FUNCTION_BLOCK LinearDA (* Basic Function Block Type *)
  (* Standard: 61499-2 *)
  (* Version 0.0, 12/23/2020, midhu, nxtControl GmbH, Template *)
  PACKAGE Main;
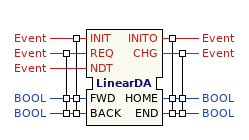
  EVENT_INPUT
    INIT WITH FWD, BACK;
    REQ WITH FWD, BACK; (* Initialization Request *)
    NDT; (* Non deterministic transition *)
  END_EVENT
  EVENT_OUTPUT
    INITO WITH HOME, END;
    CHG WITH HOME, END; (* Initialization Confirm *)
  END_EVENT
  VAR_INPUT
    FWD : BOOL; (* Input event qualifier *)
    BACK : BOOL;
  END_VAR
  VAR_OUTPUT
    HOME : BOOL; (* Output event qualifier *)
    END : BOOL;
  END_VAR
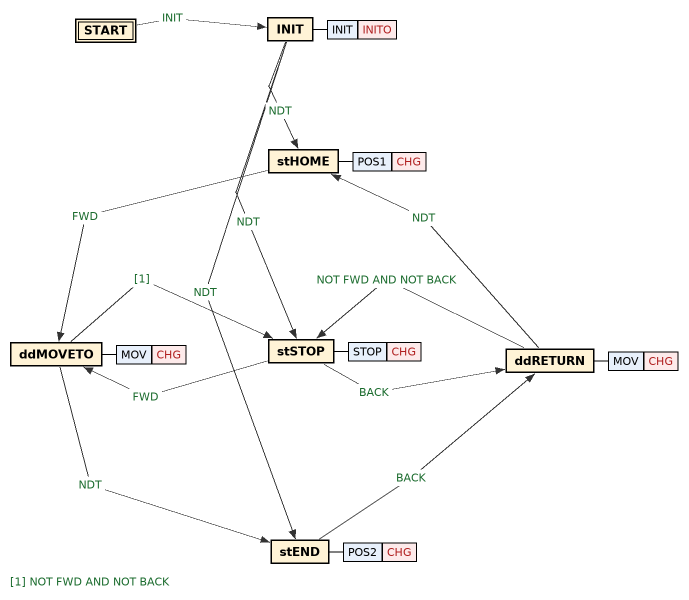
  EC_STATES
    START; (* Initial State *)
    INIT : INIT -> INITO; (* Initialization *)
    stHOME : POS1 -> CHG;
    stEND : POS2 -> CHG;
    ddMOVETO : MOV -> CHG;
    ddRETURN : MOV -> CHG;
    stSTOP : STOP -> CHG;
  END_STATES
  EC_TRANSITIONS
    START TO INIT := INIT;
    INIT TO stHOME := NDT;
    stHOME TO ddMOVETO := FWD;
    stEND TO ddRETURN := BACK;
    ddMOVETO TO stEND := NDT;
    ddRETURN TO stHOME := NDT;
    ddRETURN TO stSTOP := NOT FWD AND NOT BACK;
    stSTOP TO ddRETURN := BACK;
    stSTOP TO ddMOVETO := FWD;
    ddMOVETO TO stSTOP := NOT FWD AND NOT BACK;
    INIT TO stSTOP := NDT;
    INIT TO stEND := NDT;
  END_TRANSITIONS
  ALGORITHM INIT IN ST: (* Initialization algorithm *)
HOME  :=TRUE;
END   :=FALSE;
  END_ALGORITHM
  ALGORITHM POS1 IN ST:
HOME  :=TRUE;
END   :=FALSE;
  END_ALGORITHM
  ALGORITHM POS2 IN ST:
HOME  :=FALSE;
END   :=TRUE;
  END_ALGORITHM
  ALGORITHM MOV IN ST:
HOME  :=FALSE;
END   :=FALSE;
  END_ALGORITHM
  ALGORITHM STOP IN ST:
HOME  :=FALSE;
END   :=FALSE;
  END_ALGORITHM
END_FUNCTION_BLOCK
